ABB RAPID module: Wobj_miwobj.mod

MODULE Wobj_miwobj
	! Points are read in order of declaration.
  ! Please do not change the order of points!

  LOCAL PERS robtarget pWobj_U_PointX1:=[[-212.3124,584.9694,6.180584],[0.0255002565681934,0.989425361156464,0.142785251140594,0.000469017511932179],[1,-2,0,0],[9E+09,9E+09,9E+09,9E+09,9E+09,9E+09]];
	LOCAL PERS robtarget pWobj_U_PointX2:=[[-114.2873,584.9677,-1.644611],[0.0254992675036192,0.989420890808105,0.142816096544266,0.000487014127429575],[1,-3,1,0],[9E+09,9E+09,9E+09,9E+09,9E+09,9E+09]];
	LOCAL PERS robtarget pWobj_U_PointY1:=[[-211.6136,441.6516,8.804858],[0.0205782279372215,0.940452635288239,-0.265419691801071,-0.211372435092926],[1,-2,1,0],[9E+09,9E+09,9E+09,9E+09,9E+09,9E+09]];

ENDMODULE
